TYPE ST_HomeOutputs :
STRUCT
    DummyRoom : ST_DummyRoomOutputs;
END_STRUCT
END_TYPE

(* stored: Version 1.1.0.1
   DUT ST_HomeOutputs: Id {d9d0aa6c-92c9-448e-8a2d-c05d1f979c07} *)
